TEXTLIST StationList_TextList
  0 = 'Process'
  1 = 'Decision'
   = ''
END_TEXTLIST

(* stored: Version 1.1.0.1, ProductVersion 3.1.4024.12
   TextList StationList_TextList: Id {5f915d7f-6102-4070-9217-3628beea02cf} *)
